{attribute addProperty BoxType "EL6201-0000-0017"}
{attribute addProperty Id "Slave_22A_DO0BIT10.125169Slave_22A_DO1BIT10.125170Slave_22A_DO2BIT10.125171Slave_22A_DO3BIT10.125172Slave_22B_DO0BIT10.125173Slave_22B_DO1BIT10.125174Slave_22B_DO2BIT10.125175Slave_22B_DO3BIT10.125176"}
{attribute addProperty CRC "730044701"}
{attribute addProperty SizeInBites "8"}
{attribute addProperty SizeInBytes "1"}
TYPE Slave_22_Outputs_2B83991D :
STRUCT
	{attribute addProperty Name "Slave_22A_DO0"}
	Slave_22A_DO0 : BIT;
	{attribute addProperty Name "Slave_22A_DO1"}
	Slave_22A_DO1 : BIT;
	{attribute addProperty Name "Slave_22A_DO2"}
	Slave_22A_DO2 : BIT;
	{attribute addProperty Name "Slave_22A_DO3"}
	Slave_22A_DO3 : BIT;
	{attribute addProperty Name "Slave_22B_DO0"}
	Slave_22B_DO0 : BIT;
	{attribute addProperty Name "Slave_22B_DO1"}
	Slave_22B_DO1 : BIT;
	{attribute addProperty Name "Slave_22B_DO2"}
	Slave_22B_DO2 : BIT;
	{attribute addProperty Name "Slave_22B_DO3"}
	Slave_22B_DO3 : BIT;
END_STRUCT
END_TYPE

(* stored: Version 1.2.0.0, ProductVersion 3.1.4024.9
   DUT Slave_22_Outputs_2B83991D: Id {6aef0d17-ca5b-4518-ae15-c590f958e69c} *)
